// TIA Portal V20 export
DATA_BLOCK "DB_Axis"   // DB410
// stored: AutoNumber false, InstanceOfName FB_Axis, InstanceOfType FB
"FB_Axis"
   // VAR
   //    "sBrakeTest ZM" { S7_SetPoint := 'True'} : "FB_BrakeTest";
   //    "sBrakeTest ZL" { S7_SetPoint := 'True'} : "FB_BrakeTest";
   //    "BrakeTest ZM" : Struct
   //       sSBTDone { S7_SetPoint := 'True'} : Bool;
   //       sStartSBT { S7_SetPoint := 'True'} : Bool;
   //       sDone { S7_SetPoint := 'True'} : Bool;
   //       sError : Bool;
   //       sStateNum : Int;
   //       sDiagnoseError : Int;
   //       scloseExternalBrake : Bool;
   //    END_STRUCT;
   //    "BrakeTest ZL" : Struct
   //       sSBTDone { S7_SetPoint := 'True'} : Bool;
   //       sStartSBT { S7_SetPoint := 'True'} : Bool;
   //       sDone { S7_SetPoint := 'True'} : Bool;
   //       sError : Bool;
   //       sStateNum : Int;
   //       sDiagnoseError : Int;
   //       scloseExternalBrake : Bool;
   //    END_STRUCT;
   //    sErrorN : Array[1..8] of Bool;
   //    sTestStopRequested : Bool;
   //    sTestStopStart : Bool;
   //    sTestStopError : Bool;
   //    sTestStopEnd : Bool;
   //    sTestStopDone : Bool;
   //    sLedSITestOK : Bool;
   //    sLedSITestSlowFlashing : Bool;
   //    sLedSITestQuickFlashing : Bool;
   //    sTimerTestStopStart : TON_TIME;
   //    sTimerTestStopEnd : TON_TIME;
   // END_VAR
   // VAR RETAIN
   //    DisableAxis01_X { S7_SetPoint := 'True'} : Bool;
   //    DisableAxis02_Y { S7_SetPoint := 'True'} : Bool;
   //    DisableAxis03_ZM { S7_SetPoint := 'True'} : Bool;
   //    DisableAxis04_B { S7_SetPoint := 'True'} : Bool;
   //    DisableAxis05_U1 { S7_SetPoint := 'True'} : Bool;
   //    DisableAxis06_U2 { S7_SetPoint := 'True'} : Bool;
   //    DisableAxis07_V { S7_SetPoint := 'True'} : Bool;
   //    DisableAxis08_W { S7_SetPoint := 'True'} : Bool;
   //    DisableAxis09_ZL { S7_SetPoint := 'True'} : Bool;
   // END_VAR
BEGIN
END_DATA_BLOCK
